// IEEE-754 classification by integer exponent bits; no floating-point operation.
// Safe with runtime floating-point exceptions enabled, including signaling NaNs.
FUNCTION F_IsFiniteLReal : BOOL
VAR_INPUT value : LREAL; END_VAR
VAR bits : LWORD; END_VAR

Tc2_System.MEMCPY(destAddr := ADR(bits), srcAddr := ADR(value), n := SIZEOF(bits));
F_IsFiniteLReal := (bits AND LWORD#16#7FF0000000000000) <> LWORD#16#7FF0000000000000;

END_FUNCTION

(* stored: Version 1.1.0.1
   POU F_IsFiniteLReal: Id {e99e098c-d348-4bae-883d-35f396b7f476} *)
